{attribute 'qualified_only'}
VAR_GLOBAL
	bVar1	: BOOL;
	iVar1: DINT;
END_VAR

(* stored: Version 1.1.0.1, ProductVersion 3.1.4024.9
   GVL DataExchange: Id {5efe0d96-5a4c-463c-a6f6-696f65a50846} *)
